TYPE UNIFIED_PROGRAM_CONFIGURATION :
STRUCT
	Name : STRING(255) := 'New program';
	Version : DATE_AND_TIME;
	Steps : ARRAY [0..UnifiedProgramConstants.MaxStepCount - 1] OF UNIFIED_PROGRAM_STEP;
END_STRUCT
END_TYPE

(* stored: Version 1.1.0.1
   DUT UNIFIED_PROGRAM_CONFIGURATION: Id {3262a4b8-794f-4cef-9c39-7eaa78c15c66} *)
